TYPE ST_CELL :
STRUCT
	Cmd : E_CMD_CELL;
	PlaceObject : BOOL; 
END_STRUCT
END_TYPE

(* stored: Version 1.1.0.1, ProductVersion 3.1.4024.12
   DUT ST_CELL: Id {fff95e0f-584d-4dcb-9bf7-5d06d476d2f2} *)
